{attribute 'no_check'}
FUNCTION_BLOCK EAP_DEVICE_IO 
VAR_OUTPUT CONSTANT
END_VAR
VAR_INPUT
	{attribute 'displaymode':='hex'}
	DevCtrl				AT %Q*:	UINT;
END_VAR		
VAR_OUTPUT	
	{attribute 'displaymode':='hex'}
	DevState			AT %I*:	UINT;
	
	LinkError				:	BOOL; //0x0001 = Link error
	IOLockedAfterLinkErr	:	BOOL; //0x0002 = I/O locked after link error (I/O reset required)
	OutOfSendResources		:	BOOL; //0x0010 = Out of send resources (I/O reset required)
	WatchdogTriggered		:	BOOL; //0x0020 = Watchdog triggered
	EthMiniportNotFound		:	BOOL; //0x0040 = Ethernet driver (miniport) not found
	ResetActive				:	BOOL; //0x0080 = I/O reset active
END_VAR
VAR
END_VAR

	(* IOs 									*)
	(****************************************)

(* Read status *****************************************)
	LinkError				:= DevState.0;
	IOLockedAfterLinkErr	:= DevState.1;
	
	OutOfSendResources		:= DevState.4;
	WatchdogTriggered		:= DevState.5;
	EthMiniportNotFound		:= DevState.6;
	ResetActive				:= DevState.7;
	
(*******************************************************)

PROPERTY PUBLIC resetRequired : bool
GET
resetRequired := IOLockedAfterLinkErr or OutOfSendResources;
END_GET
END_PROPERTY

END_FUNCTION_BLOCK

(* stored: Version 1.1.0.1, ProductVersion 3.1.4024.15
   POU EAP_DEVICE_IO: Id {83f9d910-7cb0-44e4-95c1-828b6e16d7e8}, SpecialFunc None
   Property resetRequired: Id {ecdb5b1f-95cb-4895-9843-7fba7958dc92}
   Get Get: Id {976d5b73-9e68-441f-b57e-549c76598fbe} *)
